{attribute 'linkalways'} 
{attribute 'no_explicit_call' := 'This FB is a CLASS and must be accessed using methods or properties'}
{attribute 'enable_dynamic_creation'}
FUNCTION_BLOCK FINAL NOT_LINT EXTENDS Node
VAR
	in : _LINT(0);
	out : _LINT(0);
END_VAR

METHOD PUBLIC Clone : I_Node
VAR
	pNode : POINTER TO NOT_LINT;
END_VAR
pNode := __NEW(NOT_LINT);
Clone := pNode^;
END_METHOD

METHOD FB_init : BOOL
VAR_INPUT
	bInitRetains : BOOL; // if TRUE, the retain variables are initialized (warm start / cold start)
	bInCopyCode : BOOL;  // if TRUE, the instance afterwards gets moved into the copy code (online change)
END_VAR
AddInput('in',THIS^.in);
AddOutput('out', THIS^.out);
END_METHOD

METHOD PROTECTED OnExecute
VAR
END_VAR
out.Value := NOT in.Value;
END_METHOD

END_FUNCTION_BLOCK

(* stored: Version 1.1.0.1, ProductVersion 3.1.4024.15
   POU NOT_LINT: Id {bff379b9-0c82-4704-bef9-ce7100304e72}, SpecialFunc None
   Folder Constructor: Id {4cc4133a-cd51-4dc0-8cf0-4131788d99f8}
   Method Clone: Id {26cbc81e-8881-4ec6-acc7-c14c89796e2a}
   Method FB_init: Id {3299c249-b207-4760-9d23-3b32799c8352}
   Method OnExecute: Id {626f624e-7432-4052-8cf7-ce7ff5f24902} *)
